# B&R Automation Studio project MappAssetInt
Automation Studio 4.12.9.18 SP; technology packages: mapp 5.24.2

## Configuration X20CP

CPU X20CP3687X, AutomationRuntime 6.7.6, Build 11.3.0, Safety 0.0, Vc 6.0.0

### Task classes (Cpu.sw)
```
Cyclic#8:
  AssetTest <- AssetTest.prg
  Sample <- exAssetInt.Sample.prg
  Shift <- Shift.prg
VcDataObjects: Vis <- Vis.dob
Binaries: vcnet, udbdef, vcrt, vcpkat, vcctext, vctcal, vcfile, vcgclass, vccstr, vcpdsw, arial, vcdsint, vcmgr, vcdsloc, vcfntttf, vccovl, vcshared, arialbd, vcalarm, vccdt, vcpdvnc, vcpfar00, vcbclass, TCData, vccnum, arsvcreg, vccshape, vccbtn, vccddbox, Vis01, Vis02, Vis03, vcclbox, vccpopup, arconfig, User, Config, ashwd, ashwac, Role, asfw, iomap, sysconf, vcpfx20, Visu01, Visu03, Visu02, Config_1
Libraries: AsBrStr, MpData, MpBase, MpAssetInt, MpCom, FileIO, DataObj, astime, brsystem, sys_lib, runtime, standard, vcresman, asieccon, ashw, AsIODiag, exAssetInt, IecCheck
```

### Hardware
```
X20CP3687X : X20CP3687X v1.8.0.0
  Connector IF2:
    ActivateDevice = 1
    Vnc1
    VncVcObjectName1 = Vis
    VncKeyMappingFile1 = VC\PS2-Keyboard.dis
    VncRefreshRate1 = 500
    ActivateSnmp = 2
  Connector IF3:
    DNAConfiguration = manual
    CycleTime = 2000
  ConfigurationID = MappAssetInt_X20CP1583
  UserPartitionSize = 16
  UserRamSize = 731936
  RemMemSize = 300000
  TimerDeviceType = EPLX2X
  TimerDevice = X20CP3687X.IF3
  TaskClassIdleTime = 2000
  Cyclic1Duration = 2000
  Cyclic8Stack = 20000
  FileDevice1
  FileDeviceName1 = ARsim
  FileDevicePath1 = C:\Temp\AssetInt
  FileDevice2
  FileDeviceName2 = USER_HD
  FileDevicePath2 = F:\
  FtpUser1
  FtpUsername1 = admin
  FtpUserPassword1 = WA9hSMBXiqkZliudaf2dLB8I5WaEURjKd6F9iexMfBQ=
  FtpUserSalt1 = wS51ak4d
  FTPAccessRight1 = 0
  ActivateOpcUa = 1
  OpcUaInformationModels_PV_Version = 1
```

## Logical view

Binary libraries used (declarations not repeated): operator, runtime, astime, AsIecCon, sys_lib, DataObj, brsystem, FileIO, AsBrStr, standard, AsIODiag, MpBase, MpAssetInt 5.24.6, MpCom, MpData 5.24.6

### Variables.var
```iecst
(*.-.-.-.-.---------------------------------------------------------------------------------------------------------------------------------------------------------------------------------*)
VAR
	Memory : ARRAY[0..19] OF exCoreInternalRecordType;
	TmpStr1 : STRING[80];
	TmpStr2 : STRING[80];
END_VAR
(*.-.-.-.-.---------------------------------------------------------------------------------------------------------------------------------------------------------------------------------*)
VAR
	AutoCount : BOOL; (*Start auto count*)
END_VAR
VAR CONSTANT
	AutoCountCycle : UINT := 1000; (*Auto count cycle in ms*)
END_VAR
VAR
	AutoCountTime : TON_10ms;
END_VAR
(*.-.-.-.-.---------------------------------------------------------------------------------------------------------------------------------------------------------------------------------*)
VAR
	AutoCreateJobs : BOOL; (*Auto create jobs*)
	AutoCreatePieceCnt : UDINT; (*Job piece counter*)
	AutoCreateJobsCnt : UDINT; (*Job name counter*)
	AutoCreateJobsNum : {REDUND_UNREPLICABLE} UDINT := 30; (*Pieces per job auto create*)
END_VAR
(*.-.-.-.-.---------------------------------------------------------------------------------------------------------------------------------------------------------------------------------*)
VAR
	GetDateTime : BOOL;
	SetDateTime : BOOL;
	RTCtime_struct : RTCtime_typ;
END_VAR
(*.-.-.-.-.---------------------------------------------------------------------------------------------------------------------------------------------------------------------------------*)
VAR
	TestBootCounter : UDINT;
	TestResult : ARRAY[1..9] OF TestResultEnum;
	TestCase : ARRAY[1..9] OF BOOL;
	TestState : ARRAY[1..9] OF USINT;
	TestIdle : ARRAY[1..9] OF UDINT;
	TesMyId : USINT;
END_VAR
(*.-.-.-.-.---------------------------------------------------------------------------------------------------------------------------------------------------------------------------------*)
VAR
	exAssetIntCoreAdr : {REDUND_UNREPLICABLE} UDINT;
	exAssetIntCoreLen : {REDUND_UNREPLICABLE} UDINT;
	exAssetIntCore_0 : REFERENCE TO exAssetIntCore;
END_VAR
```

### Library Logical/exAssetInt/exAssetInt (IEC, version 1.50.0)

#### MpAssetInt.typ
```iecst
(*File Version 1008*)
(*------------------------------------------------------------------------------------------------------------------------------------------------------------------------------------------------------------------------------------------------------------------------------------------------------------------------------------------------------*)
(*Internal type*)

TYPE
	exCoreInternalDataType : 	STRUCT
		RecordIndexUsed : ARRAY[0..CORE_EVENT_NUM_MAX]OF BOOL; (*Next record ID*)
		RecordIndex : UINT; (*Next record ID*)
		RecordData : exCoreInternalRecordType;
		State : exAssetIntStateEnum;
		StateError : exAssetIntStateEnum := exASSETINT_STATE_NONE;
		InitAfterBoot : BOOL;
		TimeLastCallShift : TIME;
		DiffLastCallShift : UDINT;
		TimeLastCallProduction : TIME;
		DiffLastCallProduction : UDINT;
		JobPieceCounterOld : UDINT;
		JobRejectCounterOld : UDINT;
		ShiftPieceCounterOld : UDINT;
		ShiftRejectCounterOld : UDINT;
		ShiftId : SINT;
		ShiftName : STRING[20];
		TmpStr1 : STRING[500];
		TmpStr2 : STRING[50];
		Downtime : exAssetIntDowntimeEnum;
		DowntimeReason : STRING[50];
		ProductionTotalTime : UDINT;
		CurrentTime : DTGetTime;
		PowerOffTime : DATE_AND_TIME;
		TimeOfDay : TIME_OF_DAY;
		ShiftTotalTimeStart : UDINT;
		StatsRefresh : TON_10ms;
		BackupTimer : TON_10ms;
		DirCreate_0 : DirCreate;
		CreateMemory : CreateMemory;
		ReadEventData : ReadEventData;
		WriteEventData : WriteEventData;
		ReadLinkData : ReadLinkData;
		WriteLinkData : WriteLinkData;
		ExportEventData : ExportEventData;
		x : UINT;
		y : UINT;
	END_STRUCT;
	exCoreInternalRecordType : 	STRUCT
		CRC : USINT;
		FileName : STRING[80]; (*ID of the event*)
		EventType : exCoreInternalRecordEnum;
		TimeStart : DATE_AND_TIME; (*Event start*)
		TimeEnd : DATE_AND_TIME; (*Event end*)
		ShiftName : STRING[20]; (*Shift name*)
		JobName : STRING[20]; (*Job name.*)
		TotalTime : exAssetIntTimeType; (*Total time since this job started*)
		ScheduledDowntime : exAssetIntTimeType; (*Scheduled downtime since this job started*)
		UnscheduledDowntime : exAssetIntTimeType; (*Unsheduled downtime since this job started*)
		Uptime : exAssetIntTimeType; (*Uptime since this job started*)
		NominalProductionTime : exAssetIntTimeType; (*Time of production at nominal speed since this job started*)
		GoodProductionTime : exAssetIntTimeType; (*Time of good production since this job started*)
		ScheduledDowntimeRate : REAL; (*Percentage of scheduled downtime [%] since this job started*)
		UnscheduledDowntimeRate : REAL; (*Percentage of unscheduled downtime [%] since this job started*)
		NominalProductionTimeRate : REAL; (*Percentage of nominal speed running time[%] since this job started*)
		TargetPieces : UDINT; (*Specifies the target quantity of products to be produced by the machine at nominal speed*)
		TotalPieces : UDINT; (*Counter for total products since this job started*)
		GoodPieces : UDINT; (*Counter for good products since this job started*)
		RejectPieces : UDINT; (*Counter for reject products since this job started*)
		BadPieceRate : REAL; (*Percentage of bad products [%] since this job started*)
		CurrentProductionRate : REAL; (*Production rate since this job started [products / h]*)
		CurrentUser : STRING[50]; (*Currently active user*)
		AdditionalData : STRING[EVENT_ADDITONAL_DATA_LEN]; (*Additional data information*)
	END_STRUCT;
	exCoreInternalRecordEnum :
		(
		RecordTypeJob := 0,
		RecordTypeShift := 1,
		RecordTypeNoShift := 2,
		RecordTypeUptime := 3,
		RecordTypeDowntimeScheduled := 4,
		RecordTypeDowntimeUnscheduled := 5,
		RecordTypeUserChange := 6,
		RecordTypeTimeline := 10
		);
	exCoreInternalExportEnum :
		(
		ExportTypeJob,
		ExportTypeShift,
		ExportTypeTimeline
		);
	exConfigInternalDataType : 	STRUCT
		State : exAssetIntStateEnum;
		StateError : exAssetIntStateEnum := exASSETINT_STATE_NONE;
		ReadConfiguration : ReadConfiguration;
		WriteConfiguration : WriteConfiguration;
	END_STRUCT;
	exUIInternalDataType : 	STRUCT
		RecordStart : DINT; (*Visible list is starting from this index*)
		RecordCount : UINT; (*Total number of items*)
		RecordCountOld : UINT; (*Old record number is required for DESC list*)
		RecordData : exCoreInternalRecordType;
		TimeSeconds : UDINT;
		TimeLongest : UDINT;
		SortingStartTimeOld : exAssetIntUISortingEnum := exASSETINT_SORTING_ASC;
		DT_TO_DTStructure_0 : DTStructure;
		x : UDINT;
		y : UDINT;
		State : exAssetIntStateEnum;
		StateError : exAssetIntStateEnum := exASSETINT_STATE_NONE;
	END_STRUCT;
	exAssetIntLinkType : 	STRUCT
		Version : USINT; (*Data structure version*)
		MemoryDb : UDINT; (*Database memory*)
		MemoryJob : UDINT; (*Job data memory*)
		MemoryShift : UDINT; (*Shift data memory*)
		MemoryTimeline : UDINT; (*Timeline data memory*)
		StatsLastCall : DTStructure; (*Date and time when the stats were last calculated*)
		Configuration : exAssetIntCoreConfigType; (*Configuration structure*)
		RecordCount : UINT; (*Number of total records*)
		IsCoreActive : BOOL; (*Core function block is ready*)
		RefreshJobUI : BOOL; (*Update job stats in UI*)
		RefreshShiftUI : BOOL; (*Update shift stats in UI*)
		RefreshTimelineUI : BOOL; (*Update timeline stats in UI*)
		ShiftStatistics : exAssetIntShiftStatisticsType; (*Current shift stats*)
		ShiftTotalTime : LREAL; (*Milliseconds the job is running*)
		ShiftDowntimeScheduled : UDINT; (*Milliseconds of scheduled downtime*)
		ShiftDowntimeUnscheduled : UDINT; (*Milliseconds of unscheduled downtime*)
		ShiftSecondsToEnd : UDINT;
		JobStatistics : exAssetIntJobStatisticsType; (*Current job stats*)
		JobTotalTime : LREAL; (*Milliseconds the job is running*)
		JobDowntimeScheduled : UDINT; (*Milliseconds of scheduled downtime*)
		JobDowntimeUnscheduled : UDINT; (*Milliseconds of unscheduled downtime*)
		ShiftId : SINT := -1; (*Index of shift configuration*)
		ProductionStateStart : DATE_AND_TIME; (*Current state beginning*)
		ProductionState : exAssetIntUIProductionStateEnum; (*Current state*)
		ProductionTotalTime : LREAL; (*Milliseconds the state is running*)
		ProductionUserName : STRING[50]; (*Currently active user*)
		ProductionShiftName : STRING[20]; (*ShiftName for this timeline*)
		ProductionJobName : STRING[20]; (*Job name for this timeline*)
		ProductionDowntime : exAssetIntDowntimeEnum; (*Downtime for this timeline*)
		ProductionDowntimeReason : STRING[50]; (*Donwtime reason for this timeline*)
	END_STRUCT;
END_TYPE

(*Enum type*)

TYPE
	exAssetIntStateEnum :
		(
		exASSETINT_STATE_INIT_1 := 1, (*Init state*)
		exASSETINT_STATE_INIT_2 := 2, (*Init state*)
		exASSETINT_STATE_INIT_3 := 3, (*Init state*)
		exASSETINT_STATE_INIT_4 := 4, (*Init state*)
		exASSETINT_STATE_INIT_5 := 5, (*Init state*)
		exASSETINT_STATE_IDLE := 10, (*Wait for command and collect data*)
		exASSETINT_STATE_STORE_EVENT := 20, (*Store new event data*)
		exASSETINT_STATE_EXPORT_EVENTS := 21, (*Export all events*)
		exASSETINT_STATE_UI_BUFFER := 30, (*Copy job data from global buffer to UI buffer*)
		exASSETINT_STATE_UI_DATA := 31, (*Generate UI data*)
		exASSETINT_STATE_SAVE_CFG := 40, (*Save configuration*)
		exASSETINT_STATE_LOAD_CFG := 41, (*Load configuration*)
		exASSETINT_STATE_SAVE_LINK := 50, (*Save internal data*)
		exASSETINT_STATE_LOAD_LINK := 51, (*Load internal data*)
		exASSETINT_STATE_ERROR := 90, (*Error state*)
		exASSETINT_STATE_NONE := 99 (*Empty state*)
		);
	exAssetIntLogLevelEnum :
		(
		exASSETINT_LOG_OFF := 0, (*Logging is disabled*)
		exASSETINT_LOG_ERROR := 1, (*Only log errors*)
		exASSETINT_LOG_INFO := 2, (*Also log information*)
		exASSETINT_LOG_ALL := 3 (*Log everything*)
		);
	exAssetIntBufferOffsets :
		(
		exASSETINT_BUFFER_MEMORY := 0
		);
	exAssetIntUIStatusEnum :
		(
		exASSETINT_UI_STATUS_IDLE := 0, (*Status: Idle, Waiting for command*)
		exASSETINT_UI_STATUS_UPDATE := 1, (*Status: Updating UIConnect structer*)
		exASSETINT_UI_STATUS_FILTER := 2 (*Status: Showing filter-dialog*)
		);
	exAssetIntMemoryEnum :
		(
		exASSETINT_MEM_DB := 0, (*Database memory*)
		exASSETINT_MEM_JOB := 1, (*Job working memory*)
		exASSETINT_MEM_SHIFT := 2, (*Shift working memory*)
		exASSETINT_MEM_TIMELINE := 3 (*Timeline working memory*)
		);
	exAssetIntDowntimeEnum :
		(
		exASSETINT_NO_DOWNTIME := 0, (*No downtime active = uptime*)
		exASSETINT_SCHEDULED_DOWNTIME := 1, (*Additional scheduled downtime (e.g. monthly maintenance)*)
		exASSETINT_UNSCHEDULED_DOWNTIME := 2 (*Unscheduled downtime (e.g. machine fault)*)
		);
	exComSeveritiesEnum :
		(
		exCOM_SEV_SUCCESS := 0, (*Success - no error*)
		exCOM_SEV_INFORMATIONAL := 1, (*Severity: Informational*)
		exCOM_SEV_WARNING := 2, (*Severity: Warning*)
		exCOM_SEV_ERROR := 3 (*Severity: Error*)
		);
END_TYPE

(*Config type*)

TYPE
	exAssetIntCoreConfigType : 	STRUCT
		CalculationTimeBase : UDINT := 1000; (*Cycle time for calculating the current production rate*)
		Shifts : ARRAY[0..4]OF exAssetIntShiftParType := [5(0)]; (*Shift schedule in detailed*)
		Export : exAssetIntExportType; (*Configuration for export*)
	END_STRUCT;
	exAssetIntExportType : 	STRUCT
		JobStatistics : BOOL := TRUE; (*Export the job statistics or not.*)
		JobStatisticsFileNamePattern : STRING[50] := 'JobStatistics_%Y_%m_%d_%H_%M.csv'; (*Pattern for export job statistics file.*)
		ShiftStatistics : BOOL := TRUE; (*Export the shift statistics or not.*)
		ShiftStatisticsFileNamePattern : STRING[50] := 'ShiftStatistics_%Y_%m_%d_%H_%M.csv'; (*Pattern for export shift statistics file.*)
		Timeline : BOOL := TRUE; (*Export the timeline statistics or not.*)
		TimelineFileNamePattern : STRING[50] := 'Timeline_%Y_%m_%d_%H_%M.csv'; (*Pattern for export timeline  file.*)
		TimestampPattern : STRING[50] := '%Y-%m-%d %H:%M:%S'; (*Timestamp pattern in exported file.*)
		DecimalDigits : UINT := 2; (*Specifies how many decimal positions are saved*)
		ColumnSeparator : STRING[1] := ','; (*Delimiter used to split up PVs in the .csv file*)
		DecimalMark : STRING[1] := '.'; (*Character to be used for the decimal separator*)
	END_STRUCT;
	exAssetIntShiftParType : 	STRUCT
		Name : STRING[20]; (*Shift name*)
		TotalTime : exAssetIntTimeSlotType; (*Total time of one shift*)
		ScheduledDowntime : ARRAY[0..9]OF exAssetIntScheduledDowntimeType; (*Scheduled downtime in one shift*)
	END_STRUCT;
	exAssetIntTimeSlotType : 	STRUCT
		Start : TIME_OF_DAY; (*Start time.*)
		End : TIME_OF_DAY; (*End time*)
	END_STRUCT;
	exAssetIntScheduledDowntimeType : 	STRUCT
		Reason : STRING[50]; (*Downtime reason*)
		Start : TIME_OF_DAY; (*Start time.*)
		End : TIME_OF_DAY; (*End time*)
	END_STRUCT;
END_TYPE

(*Parameter type*)

TYPE
	exAssetIntParType : 	STRUCT
		NominalProductionRate : REAL := 0.0; (*Nominal production rate [products / h]*)
		Job : STRING[20] := 'Job1'; (*Currently active production job*)
		CurrentUser : STRING[50]; (*Currently logged in user*)
		AdditionalData : STRING[255]; (*Additional data to be logged*)
	END_STRUCT;
END_TYPE

(*UI type*)

TYPE
	exAssetIntUITrendType : 	STRUCT
		SaexleData : ARRAY[0..365]OF REAL; (*FB->VC:Saexle data for trend data*)
		SaexleRate : UDINT; (*FB->VC:Saexle rate datapoint for trend data*)
		SaexleCount : UDINT; (*FB->VC:Saexle count datapoint for trend data*)
		SaexleDateTime : DATE_AND_TIME; (*FB->VC:Saexle DataTime datapoint for trend data*)
		MinValue : REAL; (*FB->VC:Min.value datapoint for trend data*)
		MaxValue : REAL; (*FB->VC:Max.value datapoint for trend data*)
		HideCurve : INT; (*FB->VC:Hide the curve if set to 1, status datapoint for trend curve*)
		TimeZoom : REAL; (*FB->VC:Zoom datapoint for trend time scale.*)
		TimeScroll : REAL; (*FB->VC:Scoll datapoint for trend time scale.*)
	END_STRUCT;
	exAssetIntUIShiftListType : 	STRUCT
		ShiftNames : ARRAY[0..5]OF STRING[20]; (*FB->VC: Shift names, *)
		SelectedIndex : UINT; (*VC->FB: Selection index for ShiftList.*)
		MaxSelection : USINT;
	END_STRUCT;
	exAssetIntTrendUIConnectType : 	STRUCT
		Status : exAssetIntUIStatusEnum; (*Status of UI function block*)
		ScheduledDowntimeRate : exAssetIntUITrendType; (*Trend for scheduled downtime rate*)
		UnscheduledDowntimeRate : exAssetIntUITrendType; (*Trend for unscheduled downtime rate*)
		NominalProductionRate : exAssetIntUITrendType; (*Trend for nominal production rate*)
		BadPieceRate : exAssetIntUITrendType; (*Trend for bad piece rate*)
		ShiftList : exAssetIntUIShiftListType; (*Determine which shift in the day is shown in the trend*)
		Filter : exAssetIntUIFilterType; (*Output filter.*)
	END_STRUCT;
	exAssetIntUITimelineOutputType : 	STRUCT
		StartTime : ARRAY[0..UI_TIMELINE_IDX]OF DATE_AND_TIME; (*FB->VC:Start time of this state*)
		ShiftName : ARRAY[0..UI_TIMELINE_IDX]OF STRING[20]; (*FB->VC:Shift name*)
		JobName : ARRAY[0..UI_TIMELINE_IDX]OF STRING[20]; (*FB->VC:Job name*)
		ProductionState : ARRAY[0..UI_TIMELINE_IDX]OF exAssetIntUIProductionStateEnum; (*FB->VC:Production state*)
		Reason : ARRAY[0..UI_TIMELINE_IDX]OF STRING[50]; (*FB->VC:Reason of this state*)
		Duration : ARRAY[0..UI_TIMELINE_IDX]OF exAssetIntTimeType; (*FB->VC:Duration of this state*)
		DurationBar : ARRAY[0..UI_TIMELINE_IDX]OF exAssetIntUITimeBargraphType; (*FB->VC:Duration of this state in a graphic way*)
		RangeStart : REAL; (*Displayed range: Start %*)
		RangeEnd : REAL; (*Displayed range: End %*)
		PageUp : BOOL; (*Command: Page Up (Scroll Up)*)
		StepUp : BOOL; (*Command: Line Up (Scroll Up)*)
		StepDown : BOOL; (*Command: Line Down (Scroll Down)*)
		PageDown : BOOL; (*Command: Page Down (Scroll Down)*)
	END_STRUCT;
	exAssetIntUITimeBargraphType : 	STRUCT
		Duration : UDINT; (*FB->VC:EndValue(lenth) of the scale*)
		Color : UDINT; (*FB->VC:ColorDatapoint of the scale*)
	END_STRUCT;
	exAssetIntTimelineUIConnectType : 	STRUCT
		Status : exAssetIntUIStatusEnum; (*Status of UI function block*)
		Output : exAssetIntUITimelineOutputType; (*Output information.*)
		Filter : exAssetIntUIFilterType; (*Output filter.*)
	END_STRUCT;
	exAssetIntTimeType : 	STRUCT
		Hours : UDINT; (*Numbers of hours*)
		Minutes : USINT; (*Numbers of minutes within an hour*)
		Seconds : USINT; (*Numbers of seconds within a minute*)
	END_STRUCT;
	exAssetIntShiftListUIConnectType : 	STRUCT
		Status : exAssetIntUIStatusEnum; (*Status of UI function block*)
		Output : exAssetIntUIShiftListOutputType; (*Output information.*)
		Filter : exAssetIntUIFilterType; (*Output filter.*)
	END_STRUCT;
	exAssetIntUIShiftListOutputType : 	STRUCT
		StartTime : ARRAY[0..UI_SHIFT_LIST_IDX]OF DATE_AND_TIME; (*Start time list*)
		EndTime : ARRAY[0..UI_SHIFT_LIST_IDX]OF DATE_AND_TIME; (*End time list*)
		ShiftName : ARRAY[0..UI_SHIFT_LIST_IDX]OF STRING[20]; (*Shift ID list*)
		CurrentUser : ARRAY[0..UI_SHIFT_LIST_IDX]OF STRING[50]; (*Currently active user*)
		AdditionalData : ARRAY[0..UI_SHIFT_LIST_IDX]OF STRING[255]; (*Additional data information*)
		TargetPieces : ARRAY[0..UI_SHIFT_LIST_IDX]OF UDINT; (*Target pieces list*)
		TotalPieces : ARRAY[0..UI_SHIFT_LIST_IDX]OF UDINT; (*Total pieces list*)
		GoodPieces : ARRAY[0..UI_SHIFT_LIST_IDX]OF UDINT; (*Good pieces list*)
		RejectPieces : ARRAY[0..UI_SHIFT_LIST_IDX]OF UDINT; (*Reject pieces list*)
		BadPieceRate : ARRAY[0..UI_SHIFT_LIST_IDX]OF REAL; (*bad piece rate list*)
		TotalTime : ARRAY[0..UI_SHIFT_LIST_IDX]OF exAssetIntTimeType; (*Total time list*)
		ScheduledDowntime : ARRAY[0..UI_SHIFT_LIST_IDX]OF exAssetIntTimeType; (*Scheduled Downtime list*)
		UnscheduledDowntime : ARRAY[0..UI_SHIFT_LIST_IDX]OF exAssetIntTimeType; (*Unscheduled Downtime list*)
		Uptime : ARRAY[0..UI_SHIFT_LIST_IDX]OF exAssetIntTimeType; (*Uptime list*)
		GoodProductionTime : ARRAY[0..UI_SHIFT_LIST_IDX]OF exAssetIntTimeType; (*Good production time list*)
		NominalProductionTime : ARRAY[0..UI_SHIFT_LIST_IDX]OF exAssetIntTimeType; (*nominal production time list*)
		NominalProductionRate : ARRAY[0..UI_SHIFT_LIST_IDX]OF REAL; (*nominal production rate list*)
		ShiftProductionRate : ARRAY[0..UI_SHIFT_LIST_IDX]OF REAL; (*Shift production rate list*)
		ScheduledDowntimeRate : ARRAY[0..UI_SHIFT_LIST_IDX]OF REAL; (*scheduled downtime rate list*)
		UnscheduledDowntimeRate : ARRAY[0..UI_SHIFT_LIST_IDX]OF REAL; (*unscheduled downtime rate list*)
		ProductionRate : ARRAY[0..UI_SHIFT_LIST_IDX]OF REAL; (*current production rate list*)
		RangeStart : REAL; (*Displayed range: Start %*)
		RangeEnd : REAL; (*Displayed range: End %*)
		PageUp : BOOL; (*Command: Page Up (Scroll Up)*)
		StepUp : BOOL; (*Command: Line Up (Scroll Up)*)
		StepDown : BOOL; (*Command: Line Down (Scroll Down)*)
		PageDown : BOOL; (*Command: Page Down (Scroll Down)*)
		IdealProductionRate : ARRAY[0..UI_SHIFT_LIST_IDX]OF REAL; (*ideal production rate list*)
		JobName : ARRAY[0..UI_SHIFT_LIST_IDX]OF STRING[20]; (*Job name list*)
	END_STRUCT;
	exAssetIntUIShiftListJobType : 	STRUCT  (*Jobs within one shift*)
		Name : ARRAY[0..9]OF STRING[20]; (*Name of the job*)
	END_STRUCT;
	exAssetIntListUISetupType : 	STRUCT
		ScrollWindow : USINT := 0; (*Scroll Window (overlap for PageUp/Down)*)
		SortingStartTime : exAssetIntUISortingEnum := exASSETINT_SORTING_DESC;
	END_STRUCT;
	exAssetIntJobListUIConnectType : 	STRUCT
		Status : exAssetIntUIStatusEnum; (*Status of UI function block*)
		Output : exAssetIntUIJobListOutputType; (*Output information.*)
		Filter : exAssetIntUIFilterType; (*Output filter.*)
	END_STRUCT;
	exAssetIntUIJobListOutputType : 	STRUCT
		JobStartTime : ARRAY[0..UI_JOB_LIST_IDX]OF DATE_AND_TIME; (*Job start time list*)
		JobEndTime : ARRAY[0..UI_JOB_LIST_IDX]OF DATE_AND_TIME; (*Job end time list*)
		JobName : ARRAY[0..UI_JOB_LIST_IDX]OF STRING[20]; (*Job name list*)
		CurrentUser : ARRAY[0..UI_JOB_LIST_IDX]OF STRING[50]; (*Currently active user*)
		AdditionalData : ARRAY[0..UI_JOB_LIST_IDX]OF STRING[255]; (*Additional data information*)
		TotalPieces : ARRAY[0..UI_JOB_LIST_IDX]OF UDINT; (*Total pieces list*)
		GoodPieces : ARRAY[0..UI_JOB_LIST_IDX]OF UDINT; (*Good pieces list*)
		RejectPieces : ARRAY[0..UI_JOB_LIST_IDX]OF UDINT; (*Reject pieces list*)
		BadPieceRate : ARRAY[0..UI_JOB_LIST_IDX]OF REAL; (*bad piece rate list*)
		TotalTime : ARRAY[0..UI_JOB_LIST_IDX]OF exAssetIntTimeType; (*Total time list*)
		ScheduledDowntime : ARRAY[0..UI_JOB_LIST_IDX]OF exAssetIntTimeType; (*Scheduled Downtime list*)
		UnscheduledDowntime : ARRAY[0..UI_JOB_LIST_IDX]OF exAssetIntTimeType; (*Unscheduled Downtime list*)
		Uptime : ARRAY[0..UI_JOB_LIST_IDX]OF exAssetIntTimeType; (*Uptime list*)
		GoodProductionTime : ARRAY[0..UI_JOB_LIST_IDX]OF exAssetIntTimeType; (*Good production time list*)
		NominalProductionTime : ARRAY[0..UI_JOB_LIST_IDX]OF exAssetIntTimeType; (*nominal production time list*)
		NominalProductionRate : ARRAY[0..UI_JOB_LIST_IDX]OF REAL; (*nominal production rate list*)
		ScheduledDowntimeRate : ARRAY[0..UI_JOB_LIST_IDX]OF REAL; (*scheduled downtime rate list*)
		UnscheduledDowntimeRate : ARRAY[0..UI_JOB_LIST_IDX]OF REAL; (*unscheduled downtime rate list*)
		ProductionRate : ARRAY[0..UI_JOB_LIST_IDX]OF REAL; (*current production rate list*)
		RangeStart : REAL; (*Displayed range: Start %*)
		RangeEnd : REAL; (*Displayed range: End %*)
		PageUp : BOOL; (*Command: Page Up (Scroll Up)*)
		StepUp : BOOL; (*Command: Line Up (Scroll Up)*)
		StepDown : BOOL; (*Command: Line Down (Scroll Down)*)
		PageDown : BOOL; (*Command: Page Down (Scroll Down)*)
		ShiftName : ARRAY[0..UI_JOB_LIST_IDX]OF STRING[20]; (*Shift ID list*)
	END_STRUCT;
	exAssetIntUISortingEnum :
		(
		exASSETINT_SORTING_ASC := 0, (*Sorting ascending*)
		exASSETINT_SORTING_DESC := 1 (*Sorting descending*)
		);
	exAssetIntUIProductionStateEnum :
		(
		exASSETINT_STATE_NO_SHIFT_ACTIVE := 0, (*Inactive state*)
		exASSETINT_STATE_UPTIME := 1, (*Uptime state*)
		exASSETINT_STATE_SCHDL_DOWNTIME := 2, (*Scheduled downtime state*)
		exASSETINT_STATE_UNSCH_DOWNTIME := 3, (*Unscheduled downtime state*)
		exASSETINT_STATE_USER_CHANGE := 4 (*User change*)
		);
	exAssetIntUICurrDTFilterType : 	STRUCT
		Enable : BOOL; (*Enable Filter*)
		DateTime : DATE_AND_TIME; (*Date and time of filter*)
	END_STRUCT;
	exAssetIntUISetDTFilterType : 	STRUCT
		Enable : BOOL; (*Enable Filter*)
		Year : UINT; (*Date&Time: Year*)
		Month : USINT; (*Date&Time: Month*)
		Day : USINT; (*Date&Time: Day*)
		Hour : USINT; (*Date&Time: Hour*)
		Minute : USINT; (*Date&Time: Minute*)
	END_STRUCT;
	exAssetIntUIFilterDialogType : 	STRUCT
		LayerStatus : UINT := UI_LAYER_HIDE; (*			Filter.Dialog.LayerStatus := UI_LAYER_HIDE;
*)
		From : exAssetIntUISetDTFilterType; (*Display entries from given date&time*)
		Until : exAssetIntUISetDTFilterType; (*Display entries until given date&time*)
		Confirm : BOOL;
		Cancel : BOOL;
	END_STRUCT;
	exAssetIntUIFilterType : 	STRUCT
		ShowDialog : BOOL;
		Dialog : exAssetIntUIFilterDialogType; (*Dialog-data to change filter-settings*)
		Current : exAssetIntUICurrentFilterType; (*Currently active filter settings*)
		DefaultLayerStatus : UINT;
	END_STRUCT;
	exAssetIntUICurrentFilterType : 	STRUCT
		From : exAssetIntUICurrDTFilterType; (*Starting time of current filter*)
		Until : exAssetIntUICurrDTFilterType; (*End time of current filter*)
	END_STRUCT;
END_TYPE

(*Info type*)

TYPE
	exAssetIntJobStatisticsType : 	STRUCT
		JobName : STRING[20]; (*Job name.*)
		StartTime : DATE_AND_TIME;
		TotalTime : exAssetIntTimeType; (*Total time since this job started*)
		ScheduledDowntime : exAssetIntTimeType; (*Scheduled downtime since this job started*)
		UnscheduledDowntime : exAssetIntTimeType; (*Unsheduled downtime since this job started*)
		Uptime : exAssetIntTimeType; (*Uptime since this job started*)
		NominalProductionTime : exAssetIntTimeType; (*Time of production at nominal speed since this job started*)
		GoodProductionTime : exAssetIntTimeType; (*Time of good production since this job started*)
		ScheduledDowntimeRate : REAL; (*Percentage of scheduled downtime [%] since this job started*)
		UnscheduledDowntimeRate : REAL; (*Percentage of unscheduled downtime [%] since this job started*)
		NominalProductionTimeRate : REAL; (*Percentage of nominal speed running time[%] since this job started*)
		TotalPieces : UDINT; (*Counter for total products since this job started*)
		GoodPieces : UDINT; (*Counter for good products since this job started*)
		RejectPieces : UDINT; (*Counter for reject products since this job started*)
		BadPieceRate : REAL; (*Percentage of bad products [%] since this job started*)
		CurrentProductionRate : REAL; (*Production rate since this job started [products / h]*)
		CurrentUser : STRING[50]; (*Currently active user*)
		AdditionalData : STRING[EVENT_ADDITONAL_DATA_LEN]; (*Additional data information*)
	END_STRUCT;
	exAssetIntShiftStatisticsType : 	STRUCT
		ShiftName : STRING[20]; (*Shift name.*)
		StartTime : DATE_AND_TIME;
		TotalTime : exAssetIntTimeType; (*Total time since this shift started*)
		ScheduledDowntime : exAssetIntTimeType; (*Scheduled downtime since this shift started*)
		UnscheduledDowntime : exAssetIntTimeType; (*Unsheduled downtime since this shift started*)
		Uptime : exAssetIntTimeType; (*Uptime since this shift started*)
		GoodProductionTime : exAssetIntTimeType; (*Time of good production since this shift started*)
		NominalProductionTime : exAssetIntTimeType; (*Time of production at nominal speed since this shift started*)
		ScheduledDowntimeRate : REAL; (*Percentage of scheduled downtime [%] since this shift started*)
		UnscheduledDowntimeRate : REAL; (*Percentage of unscheduled downtime [%] since this shift started*)
		NominalProductionTimeRate : REAL; (*Percentage of nominal speed running time[%] since this shift started*)
		TargetPieces : UDINT; (*Counter for target products since this shift started*)
		TotalPieces : UDINT; (*Counter for total products since this shift started*)
		GoodPieces : UDINT; (*Counter for good products since this shift started*)
		RejectPieces : UDINT; (*Counter for reject products since this shift started*)
		BadPieceRate : REAL; (*Percentage of bad products [%] since this shift started*)
		CurrentProductionRate : REAL; (*Production rate since this shift started [products / h]*)
		CurrentUser : STRING[50]; (*Currently active user*)
		AdditionalData : STRING[255]; (*Additional data information*)
		IdealProductionRate : REAL; (*Ideal production rate*)
	END_STRUCT;
	exAssetIntCoreInfoType : 	STRUCT
		ShiftStatistics : exAssetIntShiftStatisticsType; (*Shift statistics*)
		JobStatistics : exAssetIntJobStatisticsType; (*Job statistics*)
		Diag : exAssetIntDiagType; (*Additional diagnostic information*)
	END_STRUCT;
	exAssetIntInfoType : 	STRUCT
		Diag : exAssetIntDiagType; (*Additional diagnostic information*)
	END_STRUCT;
	exAssetIntDiagType : 	STRUCT
		StatusID : exAssetIntStatusIDType; (*Segmented StatusID output*)
	END_STRUCT;
	exAssetIntStatusIDType : 	STRUCT
		ID : exAssetIntErrorEnum; (*StatusID as enumerator*)
		Severity : exComSeveritiesEnum; (*Severity of the error*)
		Code : UINT; (*Error code*)
	END_STRUCT;
END_TYPE
```

#### Constants.var - Exported constants
```iecst
(*File Version 1007*)
(*------------------------------------------------------------------------------------------------------------------------------------------------------------------------------------------------------------------------------------------------------------------------------------------------------------------------------------------------------*)
(*General constants*)
(*------------------------------------------------------------------------------------------------------------------------------------------------------------------------------------------------------------------------------------------------------------------------------------------------------------------------------------------------------*)
VAR CONSTANT
	CORE_FOLDER_NAME : STRING[50] := 'AssetIntData'; (*Name of the event folder*)
	CORE_EVENT_NUM_MAX : UINT := 500; (*Maximum number of events*)
	CORE_BACKUP_TIMER : UINT := 10; (*Backup timer (minutes) for internal data*)
	EVENT_ADDITONAL_DATA_LEN : UINT := 100; (*Length of the event comment*)
	EXLINK_VERSION : USINT := 1; (*exLink structure version*)
END_VAR
(*------------------------------------------------------------------------------------------------------------------------------------------------------------------------------------------------------------------------------------------------------------------------------------------------------------------------------------------------------*)
(*Export constants*)
(*------------------------------------------------------------------------------------------------------------------------------------------------------------------------------------------------------------------------------------------------------------------------------------------------------------------------------------------------------*)
VAR CONSTANT
	EXPORT_BUFFER : UINT := 500; (*Length of the buffer for the event export*)
	EXPORT_JOB_TITEL : STRING[100] := 'AssetInt Job Statistics Export File'; (*Export file header*)
	EXPORT_SHIFT_TITEL : STRING[100] := 'AssetInt Shift Statistics Export File'; (*Export file header*)
	EXPORT_TIMELINE_TITEL : STRING[100] := 'AssetInt Timeline Statistics Export File'; (*Export file header*)
	EXPORT_JOB_HEADER : STRING[400] := 'Job Start Time;Job End Time;Job Name;Current User;Additional Data;Total Pieces;Good Pieces;Reject Pieces;Bad Piece Rate;Total Time;Scheduled Downtime;Unscheduled Downtime;Uptime;Good Production Time;Nominal Production Time;Nominal Production Time Rate;Scheduled Downtime Rate;Unscheduled Downtime Rate;Production Rate;Shift Name'; (*Export file column headers*)
	EXPORT_SHIFT_HEADER : STRING[400] := 'Job Start Time;Job End Time;Job Name;Current User;Additional Data;Total Pieces;Good Pieces;Reject Pieces;Bad Piece Rate;Total Time;Scheduled Downtime;Unscheduled Downtime;Uptime;Good Production Time;Nominal Production Time;Nominal Production Time Rate;Scheduled Downtime Rate;Unscheduled Downtime Rate;Production Rate;Shift Name'; (*Export file column headers*)
	EXPORT_TIMELINE_HEADER : STRING[400] := 'Start Time;Shift ID;Production State;Reason;Duration;Job Name'; (*Export file column headers*)
END_VAR
(*------------------------------------------------------------------------------------------------------------------------------------------------------------------------------------------------------------------------------------------------------------------------------------------------------------------------------------------------------*)
(*UI constants*)
(*------------------------------------------------------------------------------------------------------------------------------------------------------------------------------------------------------------------------------------------------------------------------------------------------------------------------------------------------------*)
VAR CONSTANT
	UI_SHIFT_LIST_IDX : UINT := 7; (*Max index for list box entries for shift data*)
	UI_TIMELINE_IDX : UINT := 7; (*Max index for list box entries for timeline data*)
	UI_JOB_LIST_IDX : UINT := 7; (*Max index for list box entries for job data*)
	UI_SHIFT_SHOW_JOBS : BOOL := FALSE; (*Show job changes in shift list*)
	UI_LAYER_SHOW : UINT := 0; (*Hide dialog layer*)
	UI_LAYER_HIDE : UINT := 1; (*Show dialog layer*)
	UI_LAYER_LOCK : UINT := 2; (*Lock dialog layer*)
END_VAR
(*------------------------------------------------------------------------------------------------------------------------------------------------------------------------------------------------------------------------------------------------------------------------------------------------------------------------------------------------------*)
(*Logger constants*)
(*------------------------------------------------------------------------------------------------------------------------------------------------------------------------------------------------------------------------------------------------------------------------------------------------------------------------------------------------------*)
VAR CONSTANT
	LOG_LEN : UINT := 100; (*Length of one log entry (minimum size is 50)*)
	LOG_NUM : UINT := 50; (*Number of log entries*)
	LOG_LEVEL : exAssetIntLogLevelEnum := exASSETINT_LOG_ALL; (*Define log level details*)
	CHAR_RETURN : USINT := 13; (*Carriage return*)
END_VAR
(*------------------------------------------------------------------------------------------------------------------------------------------------------------------------------------------------------------------------------------------------------------------------------------------------------------------------------------------------------*)
(*Error codes*)
(*------------------------------------------------------------------------------------------------------------------------------------------------------------------------------------------------------------------------------------------------------------------------------------------------------------------------------------------------------*)
VAR CONSTANT
	ERR_ASSET_LINK : DINT := -1064239102; (*Input exLink is 0 pointer*)
	ERR_ASSET_LINK_VERSION : DINT := 100001; (*exLink version is not compatible with backup data*)
	ERR_ASSET_LINK_SIZE : DINT := 100002; (*exLink backup data has wrong size*)
	ERR_ASSET_TEMP_MEMORY : DINT := -1064136704; (*No temporary memory available, make sure core function block is enabled*)
	ERR_ASSET_INF_WAIT_CORE_FB : DINT := 1083346949; (*This component can only become active if MpAssetIntCore is active.*)
	ERR_ASSET_READ_RECORD_SIZE : DINT := -2138009590; (*Record size is not correct during reading event data*)
	ERR_ASSET_READ_CRC : DINT := 100000; (*Record CRC error during reading event data*)
	ERR_ASSET_READ_FILE_NAME : DINT := 100003; (*File name in event folder does not match the expected event#<index> pattern*)
	ERR_ASSET_CONFIG : DINT := -1064239096; (*Configuration link is 0 pointer*)
	ERR_ASSET_CONFIG_SIZE : DINT := 100004; (*Configuration file has wrong size during reading*)
	ERR_ASSET_READ_BUFFER_FULL : DINT := 100005; (*More valid event files exist than fit into the record buffer, excess file was skipped*)
	ERR_ASSET_SHIFT_CALC : DINT := -1064239097; (*Invalid shift configured*)
END_VAR
```

#### exAssetInt.fun - Exported functions and function blocks
```iecst
(*File Version 1006*)
(*------------------------------------------------------------------------------------------------------------------------------------------------------------------------------------------------------------------------------------------------------------------------------------------------------------------------------------------------------*)

FUNCTION_BLOCK exAssetIntCore (*mapp function block which can be used for asset intensity calculation.*) (* $GROUP=mapp Services,$CAT=Asset Intensity,$GROUPICON=Icon_mapp.png,$CATICON=Icon_exOee.png *)
	VAR_INPUT
		exLink : REFERENCE TO exAssetIntLinkType; (*Incoming communication handle (mapp standard interface)*) (* *) (*#PAR#;*)
		Enable : BOOL; (*Enables/Disables the function block (mapp standard interface)*) (* *) (*#PAR#;*)
		ErrorReset : BOOL; (*Resets all function block errors (mapp standard interface)*) (* *) (*#PAR#;*)
		Parameters : REFERENCE TO exAssetIntParType; (*Function block parameters (mapp standard interface)*) (* *) (*#PAR#; *)
		Logger : UDINT;
		Configuration : REFERENCE TO exAssetIntCoreConfigType;
		Update : BOOL; (*Updates the parameters (mapp standard interface)*) (* *) (*#PAR#; *)
		Downtime : exAssetIntDowntimeEnum; (*The machine is in down time*) (* *) (*#CMD#; *)
		DowntimeReason : REFERENCE TO STRING[50]; (*The reason for down time*) (* *) (*#CMD#; *)
		PieceCounter : UDINT; (*Total pieces counter.*) (* *) (*#CMD#; *)
		RejectCounter : UDINT; (*Reject pieces counter*) (* *) (*#CMD#; *)
		DeviceName : REFERENCE TO STRING[50]; (*Address of the exported device name*) (* *) (*#CMD#; *)
		StorageName : REFERENCE TO STRING[50]; (*Address of the storage device name*) (* *) (*#CMD#; *)
		Export : BOOL; (*Export the saved information to file*) (* *) (*#CMD#; *)
		Reset : BOOL; (*Reset the data buffer*) (* *) (*#CMD#; *)
	END_VAR
	VAR_OUTPUT
		Active : BOOL; (*Function block is active (mapp standard interface)*) (* *) (*#PAR#;*)
		Error : BOOL; (*Indicates an error (mapp standard interface)*) (* *) (*#PAR#;*)
		StatusID : DINT; (*Error/Status information (mapp standard interface)*) (* *) (*#PAR#; *)
		UpdateDone : BOOL; (*Update of parameters done (mapp standard interface)*) (* *) (*#PAR#; *)
		CommandBusy : BOOL; (*Function block is busy processing a command*) (* *) (*#CMD#OPT#;*)
		CommandDone : BOOL; (*True if a command finshed successfully.*) (* *) (*#CMD#OPT#;*)
		CurrentProductionRate : REAL; (*Current production rate [products / h] based on calculation time base*) (* *) (*#CYC#*)
		ScheduledDowntimeRate : REAL; (*Percentage of scheduled downtime [%]*) (* *) (*#CYC#;*)
		UnscheduledDowntimeRate : REAL; (*Percentage of unscheduled downtime [%]*) (* *) (*#CYC#;*)
		NominalProductionTimeRate : REAL; (*Percentage of running time at nominal production speed [%]*) (* *) (*#CYC#;*)
		BadPieceRate : REAL; (*Percentage of bad products [%]*) (* *) (*#CYC#;*)
		ExportDone : BOOL; (*Export command was succesfuly finished*) (* *) (*#CMD#; *)
		Info : exAssetIntCoreInfoType; (*Provide any further useful information as function block output.(mapp standard interface)*) (* *) (*#CMD#; *)
	END_VAR
	VAR
		Internal : {REDUND_UNREPLICABLE} exCoreInternalDataType; (*Internal data*)
		zzEdge00000 : BOOL;
		zzEdge00001 : BOOL;
		zzEdge00002 : BOOL;
		zzEdge00003 : BOOL;
	END_VAR
END_FUNCTION_BLOCK

FUNCTION_BLOCK exAssetIntCoreConfig
	VAR_INPUT
		Enable : BOOL; (*Enables/Disables the function block (mapp standard interface)*) (* *) (*#PAR#;*)
		ErrorReset : BOOL; (*Resets all function block errors (mapp standard interface)*) (* *) (*#PAR#;*)
		DeviceName : REFERENCE TO STRING[30]; (*Address of the exported device name*) (* *) (*#CMD#; *)
		Configuration : REFERENCE TO exAssetIntCoreConfigType;
		Logger : UDINT;
		Load : {REDUND_UNREPLICABLE} BOOL; (* *) (* *) (*#PAR#;*)
		Save : BOOL; (* *) (* *) (*#PAR#;*)
	END_VAR
	VAR_OUTPUT
		Active : BOOL; (*Function block is active (mapp standard interface)*) (* *) (*#PAR#;*)
		Error : BOOL; (*Indicates an error (mapp standard interface)*) (* *) (*#PAR#;*)
		StatusID : DINT; (*Error/Status information (mapp standard interface)*) (* *) (*#PAR#; *)
		CommandBusy : BOOL; (*Function block is busy processing a command*) (* *) (*#CMD#OPT#;*)
		CommandDone : BOOL; (*True if a command finshed successfully.*) (* *) (*#CMD#OPT#;*)
		Info : exAssetIntInfoType; (*Provide any further useful information as function block output.(mapp standard interface)*) (* *) (*#CMD#; *)
	END_VAR
	VAR
		Internal : {REDUND_UNREPLICABLE} exConfigInternalDataType; (*Internal data*)
		zzEdge00000 : BOOL;
		zzEdge00001 : BOOL;
		zzEdge00002 : BOOL;
	END_VAR
END_FUNCTION_BLOCK

FUNCTION_BLOCK exAssetIntJobListUI (*mapp function block which can be used for showing job statistics in a list *)
	VAR_INPUT
		exLink : REFERENCE TO exAssetIntLinkType; (*Incoming communication handle (mapp standard interface)*) (* *) (*#PAR#;*)
		Enable : BOOL; (*Enables/Disables the function block (mapp standard interface)*) (* *) (*#PAR#;*)
		ErrorReset : BOOL; (*Resets all function block errors (mapp standard interface)*) (* *) (*#PAR#;*)
		Logger : UDINT;
		UISetup : exAssetIntListUISetupType; (*Setup UI connection - must be configured before enabling the FB*) (* *) (*#PAR#; *)
		UIConnect : REFERENCE TO exAssetIntJobListUIConnectType; (*Connection structure for VC4 User interface*) (* *) (*#CMD#; *)
	END_VAR
	VAR_OUTPUT
		Active : BOOL; (*Function block is active (mapp standard interface)*) (* *) (*#PAR#;*)
		Error : BOOL; (*Indicates an error (mapp standard interface)*) (* *) (*#PAR#;*)
		StatusID : DINT; (*Error/Status information (mapp standard interface)*) (* *) (*#PAR#; *)
		Info : exAssetIntInfoType; (*Provide any further useful information as function block output.(mapp standard interface)*) (* *) (*#CMD#; *)
	END_VAR
	VAR
		Internal : {REDUND_UNREPLICABLE} exUIInternalDataType; (*Internal data*)
		zzEdge00000 : BOOL;
	END_VAR
END_FUNCTION_BLOCK

FUNCTION_BLOCK exAssetIntShiftListUI (*mapp function block which can be used for showing shift statistics in a list *)
	VAR_INPUT
		exLink : REFERENCE TO exAssetIntLinkType; (*Incoming communication handle (mapp standard interface)*) (* *) (*#PAR#;*)
		Enable : BOOL; (*Enables/Disables the function block (mapp standard interface)*) (* *) (*#PAR#;*)
		ErrorReset : BOOL; (*Resets all function block errors (mapp standard interface)*) (* *) (*#PAR#;*)
		Logger : UDINT;
		UISetup : exAssetIntListUISetupType; (*Setup UI connection - must be configured before enabling the FB*) (* *) (*#PAR#; *)
		UIConnect : REFERENCE TO exAssetIntShiftListUIConnectType; (*Connection structure for VC4 User interface*) (* *) (*#CMD#; *)
	END_VAR
	VAR_OUTPUT
		Active : BOOL; (*Function block is active (mapp standard interface)*) (* *) (*#PAR#;*)
		Error : BOOL; (*Indicates an error (mapp standard interface)*) (* *) (*#PAR#;*)
		StatusID : DINT; (*Error/Status information (mapp standard interface)*) (* *) (*#PAR#; *)
		Info : exAssetIntInfoType; (*Provide any further useful information as function block output.(mapp standard interface)*) (* *) (*#CMD#; *)
	END_VAR
	VAR
		Internal : {REDUND_UNREPLICABLE} exUIInternalDataType; (*Internal data*)
		zzEdge00000 : BOOL;
	END_VAR
END_FUNCTION_BLOCK

FUNCTION_BLOCK exAssetIntTimelineUI (*mapp function block which can be used for showing timeline statistics in a list *)
	VAR_INPUT
		exLink : REFERENCE TO exAssetIntLinkType; (*Incoming communication handle (mapp standard interface)*) (* *) (*#PAR#;*)
		Enable : BOOL; (*Enables/Disables the function block (mapp standard interface)*) (* *) (*#PAR#;*)
		ErrorReset : BOOL; (*Resets all function block errors (mapp standard interface)*) (* *) (*#PAR#;*)
		Logger : UDINT;
		UISetup : exAssetIntListUISetupType; (*Setup UI connection - must be configured before enabling the FB*) (* *) (*#PAR#; *)
		UIConnect : REFERENCE TO exAssetIntTimelineUIConnectType; (*Connection structure for VC4 User interface*) (* *) (*#CMD#; *)
	END_VAR
	VAR_OUTPUT
		Active : BOOL; (*Function block is active (mapp standard interface)*) (* *) (*#PAR#;*)
		Error : BOOL; (*Indicates an error (mapp standard interface)*) (* *) (*#PAR#;*)
		StatusID : DINT; (*Error/Status information (mapp standard interface)*) (* *) (*#PAR#; *)
		Info : exAssetIntInfoType; (*Provide any further useful information as function block output.(mapp standard interface)*) (* *) (*#CMD#; *)
	END_VAR
	VAR
		Internal : {REDUND_UNREPLICABLE} exUIInternalDataType; (*Internal data*)
		zzEdge00000 : BOOL;
	END_VAR
END_FUNCTION_BLOCK

FUNCTION_BLOCK CreateMemory
	VAR_INPUT
		Enable : BOOL;
		Size : UDINT;
		Logger : {REDUND_UNREPLICABLE} UDINT; (*Address of log buffer*)
	END_VAR
	VAR_OUTPUT
		MemoryDb : UDINT;
		MemoryJob : UDINT;
		MemoryShift : UDINT;
		MemoryTimeline : UDINT;
		Status : DINT;
	END_VAR
	VAR
		DatObjCreate_0 : DatObjCreate;
		MemoryType : exAssetIntMemoryEnum;
		TmpStr1 : STRING[100];
		TmpStr2 : STRING[100];
		Cnt : USINT;
		State : USINT;
	END_VAR
END_FUNCTION_BLOCK

FUNCTION_BLOCK ReadConfiguration
	VAR_INPUT
		Enable : BOOL;
		Device : REFERENCE TO STRING[50];
		Logger : {REDUND_UNREPLICABLE} UDINT; (*Address of log buffer*)
		Configuration : exAssetIntCoreConfigType;
	END_VAR
	VAR_OUTPUT
		Status : DINT;
	END_VAR
	VAR
		FileOpen_0 : FileOpen;
		FileClose_0 : FileClose;
		FileRead_0 : FileRead;
		State : USINT;
	END_VAR
END_FUNCTION_BLOCK

FUNCTION_BLOCK WriteConfiguration
	VAR_INPUT
		Enable : BOOL;
		Device : REFERENCE TO STRING[50];
		Logger : UDINT; (*Address of log buffer*)
		Configuration : exAssetIntCoreConfigType;
	END_VAR
	VAR_OUTPUT
		Status : DINT;
	END_VAR
	VAR
		FileCreate_0 : FileCreate;
		FileOpen_0 : FileOpen;
		FileClose_0 : FileClose;
		FileWrite_0 : FileWrite;
		Ident : UDINT;
		State : USINT;
	END_VAR
END_FUNCTION_BLOCK

FUNCTION_BLOCK ReadLinkData
	VAR_INPUT
		Enable : BOOL;
		Device : REFERENCE TO STRING[50];
		Logger : {REDUND_UNREPLICABLE} UDINT;
		Link : REFERENCE TO exAssetIntLinkType;
	END_VAR
	VAR_OUTPUT
		Status : DINT;
	END_VAR
	VAR
		FileOpen_0 : FileOpen;
		FileClose_0 : FileClose;
		FileRead_0 : FileRead;
		FileDelete_0 : FileDelete;
		LinkRead : exAssetIntLinkType;
		StatusRead : DINT;
		State : USINT;
	END_VAR
END_FUNCTION_BLOCK

FUNCTION_BLOCK WriteLinkData
	VAR_INPUT
		Enable : BOOL;
		Device : REFERENCE TO STRING[50];
		Logger : UDINT;
		Link : REFERENCE TO exAssetIntLinkType;
	END_VAR
	VAR_OUTPUT
		Status : DINT;
	END_VAR
	VAR
		FileCreate_0 : FileCreate;
		FileOpen_0 : FileOpen;
		FileClose_0 : FileClose;
		FileWrite_0 : FileWrite;
		Ident : UDINT;
		State : USINT;
	END_VAR
END_FUNCTION_BLOCK

FUNCTION_BLOCK ReadEventData
	VAR_INPUT
		Enable : BOOL;
		Device : STRING[50];
		Logger : {REDUND_UNREPLICABLE} UDINT;
		Memory : UDINT;
		RecordIndexUsed : REFERENCE TO ARRAY[0..CORE_EVENT_NUM_MAX] OF BOOL;
	END_VAR
	VAR_OUTPUT
		RecordCount : UINT;
		Status : DINT;
	END_VAR
	VAR
		DirOpen_0 : DirOpen;
		DirReadEx_0 : DirReadEx;
		DirClose_0 : DirClose;
		FileOpen_0 : FileOpen;
		FileClose_0 : FileClose;
		FileRead_0 : FileRead;
		FileDelete_0 : FileDelete;
		FileName : STRING[100];
		FileInfo_0 : fiDIR_READ_EX_DATA;
		RecordData : exCoreInternalRecordType;
		FirstEntryTime : DATE_AND_TIME;
		LastEntryTime : DATE_AND_TIME;
		FirstEntryRecord : UINT;
		LastEntryRecord : UINT;
		TmpStr1 : STRING[100];
		FileIndex : UINT;
		FileIndexCheck : DINT;
		NextFileNameGet : BOOL;
		NextFileNameReady : BOOL;
		Override : {REDUND_UNREPLICABLE} USINT;
		State : USINT;
		CRC : USINT;
		StatusRead : DINT;
		zzEdge00000 : BOOL;
	END_VAR
END_FUNCTION_BLOCK

FUNCTION_BLOCK WriteEventData
	VAR_INPUT
		Enable : BOOL;
		Device : STRING[50];
		Logger : UDINT; (*Address of log buffer*)
		RecordData : UDINT;
		RecordIndex : UINT;
	END_VAR
	VAR_OUTPUT
		Status : DINT;
	END_VAR
	VAR
		FileCreate_0 : FileCreate;
		FileOpen_0 : FileOpen;
		FileClose_0 : FileClose;
		FileWrite_0 : FileWrite;
		RecordDataIntern : exCoreInternalRecordType;
		TmpStr1 : STRING[100];
		TmpStr2 : STRING[10];
		Ident : UDINT;
		State : USINT;
		zzEdge00000 : BOOL;
	END_VAR
END_FUNCTION_BLOCK

FUNCTION_BLOCK ExportEventData
	VAR_INPUT
		Enable : BOOL;
		Device : STRING[50];
		Logger : UDINT; (*Address of log buffer*)
		RecordCount : UDINT;
		Memory : UDINT;
		Configuration : exAssetIntExportType;
	END_VAR
	VAR_OUTPUT
		Status : DINT;
	END_VAR
	VAR
		ExportType : exCoreInternalExportEnum;
		FileDelete_0 : FileDelete;
		FileCreate_0 : FileCreate;
		FileClose_0 : FileClose;
		FileWrite_0 : FileWrite;
		RtcGettime : {REDUND_UNREPLICABLE} RTCtime_typ;
		RecordDataIntern : exCoreInternalRecordType;
		DTStructure_0 : DTStructure;
		FileName : STRING[54]; (*+4 bytes to absorb %Y expansion from 2 to 4 chars*)
		TmpStr1 : STRING[54]; (*+4 bytes to absorb %Y expansion from 2 to 4 chars*)
		TmpStr2 : STRING[50];
		lrealStr : {REDUND_UNREPLICABLE} LREAL;
		Buffer : STRING[EXPORT_BUFFER];
		Offset : UDINT;
		idx : UDINT;
		State : USINT;
	END_VAR
END_FUNCTION_BLOCK

FUNCTION exAssetIntFilterListUI : UDINT
	VAR_INPUT
		Filter : REFERENCE TO exAssetIntUIFilterType;
		Status : REFERENCE TO exAssetIntUIStatusEnum;
		Logger : UDINT;
		State : exAssetIntStateEnum;
	END_VAR
	VAR
		DT_TO_DTStructure_0 : DTStructure;
	END_VAR
END_FUNCTION

FUNCTION exAssetIntScrollListUI : exAssetIntStateEnum
	VAR_INPUT
		RecordCount : UINT;
		ListMaxCount : UINT;
		PageUp : REFERENCE TO BOOL; (* *) (* *) (*#PAR#;*)
		PageDown : REFERENCE TO BOOL; (* *) (* *) (*#PAR#;*)
		StepUp : REFERENCE TO BOOL; (* *) (* *) (*#PAR#;*)
		StepDown : REFERENCE TO BOOL; (* *) (* *) (*#PAR#;*)
		RecordStart : REFERENCE TO DINT;
		RangeStart : REFERENCE TO REAL;
		RangeEnd : REFERENCE TO REAL;
		State : exAssetIntStateEnum;
	END_VAR
END_FUNCTION

FUNCTION exAssetIntBufferUI : UINT
	VAR_INPUT
		Memory : UDINT;
		exLink : exAssetIntLinkType; (*Incoming communication handle (mapp standard interface)*) (* *) (*#PAR#;*)
		SortingStartTime : exAssetIntUISortingEnum;
		Filter : exAssetIntUIFilterType;
		EventType : exCoreInternalRecordEnum;
	END_VAR
	VAR
		RecordData : exCoreInternalRecordType;
		RecordCount : UINT;
		y : UDINT;
	END_VAR
END_FUNCTION

FUNCTION exAssetIntFilterReset : BOOL
	VAR_INPUT
		Filter : REFERENCE TO exAssetIntUIFilterType;
	END_VAR
END_FUNCTION

FUNCTION exAssetIntCheckPreq : BOOL
	VAR_INPUT
		exLink : exAssetIntLinkType; (*Incoming communication handle (mapp standard interface)*) (* *) (*#PAR#;*)
		UIConnect : UDINT; (* *) (* *) (*#PAR#;*)
		Logger : UDINT;
		State : REFERENCE TO exAssetIntStateEnum;
		StatusID : REFERENCE TO DINT;
		InfoDiagStatusID : REFERENCE TO exAssetIntStatusIDType;
	END_VAR
END_FUNCTION

FUNCTION exAssetIntCheckShiftData : BOOL
	VAR_INPUT
		Configuration : exAssetIntCoreConfigType;
		Logger : UDINT;
		State : REFERENCE TO exAssetIntStateEnum;
		StatusID : REFERENCE TO DINT;
		InfoDiagStatusID : REFERENCE TO exAssetIntStatusIDType;
	END_VAR
	VAR
		TmpStr1 : STRING[100];
		TmpStr2 : STRING[100];
		y : USINT;
		x : USINT;
	END_VAR
END_FUNCTION

FUNCTION InsertEventData : USINT
	VAR_INPUT
		Memory : UDINT;
		RecordCount : UINT;
		RecordData : exCoreInternalRecordType;
	END_VAR
	VAR
		RecordMemory : REFERENCE TO exCoreInternalRecordType;
		sort : UDINT;
		x : INT;
		y : INT;
	END_VAR
END_FUNCTION

FUNCTION CreateLoggerEntry : USINT
	VAR_INPUT
		LogLevel : exAssetIntLogLevelEnum; (*Log Level*)
		LogMsg : UDINT; (*Log message*)
		LogBuffer : UDINT; (*Address of log buffer*)
	END_VAR
	VAR
		RtcGettime : RTCtime_typ;
		TmpStr : STRING[20];
		LastMsg : STRING[LOG_LEN];
		TmpMsg : STRING[LOG_LEN];
	END_VAR
END_FUNCTION

FUNCTION CreateErrorState : DINT
	VAR_INPUT
		ErrorID : DINT;
		ErrorMsg : UDINT;
		Logger : UDINT;
		Severity : exComSeveritiesEnum;
		State : REFERENCE TO exAssetIntStateEnum;
		DiagStatusID : REFERENCE TO exAssetIntStatusIDType;
	END_VAR
END_FUNCTION

FUNCTION CalcStatsJob : USINT
	VAR_INPUT
		exLink : exAssetIntLinkType; (*Incoming communication handle (mapp standard interface)*) (* *) (*#PAR#;*)
		DiffLastCall : UDINT;
		Downtime : exAssetIntDowntimeEnum;
		Parameter : exAssetIntParType;
		JobStatistics : REFERENCE TO exAssetIntJobStatisticsType;
	END_VAR
	VAR
		JobTotalTime : UDINT;
		Uptime : UDINT;
		NominalProductionTime : UDINT;
		GoodProductionTime : UDINT;
	END_VAR
END_FUNCTION

FUNCTION TrackShiftChange : BOOL
	VAR_INPUT
		exLink : REFERENCE TO exAssetIntLinkType; (*Incoming communication handle (mapp standard interface)*) (* *) (*#PAR#;*)
		Internal : REFERENCE TO exCoreInternalDataType; (*Internal data*)
		Info : REFERENCE TO exAssetIntCoreInfoType; (* *) (* *) (*#PAR#; *)
		Parameters : exAssetIntParType; (* *) (* *) (*#PAR#; *)
		Logger : UDINT;
	END_VAR
	VAR
		DiffTime : DINT;
	END_VAR
END_FUNCTION

FUNCTION TrackProductionState : BOOL
	VAR_INPUT
		exLink : REFERENCE TO exAssetIntLinkType; (*Incoming communication handle (mapp standard interface)*) (* *) (*#PAR#;*)
		Internal : REFERENCE TO exCoreInternalDataType; (*Internal data*)
		Parameters : exAssetIntParType; (* *) (* *) (*#PAR#; *)
		Logger : UDINT;
	END_VAR
END_FUNCTION

FUNCTION CalcStatsShift : USINT
	VAR_INPUT
		exLink : exAssetIntLinkType; (*Incoming communication handle (mapp standard interface)*) (* *) (*#PAR#;*)
		DiffLastCall : UDINT;
		Downtime : exAssetIntDowntimeEnum;
		Parameter : exAssetIntParType;
		ShiftStatistics : REFERENCE TO exAssetIntShiftStatisticsType;
	END_VAR
	VAR
		ShiftTotalTime : UDINT;
		Uptime : UDINT;
		NominalProductionTime : UDINT;
		GoodProductionTime : UDINT;
	END_VAR
END_FUNCTION

FUNCTION CalcCrc : USINT
	VAR_INPUT
		data : UDINT;
		length : UINT;
	END_VAR
	VAR
		idx : UINT;
		_byte : USINT;
	END_VAR
END_FUNCTION

FUNCTION FindInstr : UDINT
	VAR_INPUT
		string1 : UDINT;
		string2 : UDINT;
	END_VAR
	VAR
		idx : UDINT;
	END_VAR
END_FUNCTION

FUNCTION ReplaceString : USINT
	VAR_INPUT
		dataSTR : UDINT;
		searchSTR : UDINT;
		replaceSTR : UDINT;
	END_VAR
	VAR
		idx : UDINT;
	END_VAR
END_FUNCTION

FUNCTION ReplaceDateTime : USINT
	VAR_INPUT
		dataSTR : UDINT;
		searchSTR : UDINT;
		value : UINT;
	END_VAR
	VAR
		lrealStr : LREAL;
	END_VAR
END_FUNCTION

FUNCTION NormalizeDateTime : LREAL
	VAR_INPUT
		value : UDINT;
	END_VAR
	VAR
		TmpStr1 : STRING[6] := '';
		TmpStr2 : STRING[6] := '';
	END_VAR
END_FUNCTION

FUNCTION NormalizeFloat : LREAL
	VAR_INPUT
		value : REAL;
		output : UDINT;
		configuration : exAssetIntExportType;
	END_VAR
	VAR
		idx : UDINT;
		tmpStr : STRING[50];
	END_VAR
END_FUNCTION
```

#### exAssetIntCore.st
```iecst
// -------------------------------------------------------------------------------------------
// File version 1013
// -------------------------------------------------------------------------------------------
// Core function block
FUNCTION_BLOCK exAssetIntCore
	// -------------------------------------------------------------------------------------------
	// Reset everything when enable is false
	IF NOT Enable THEN
		Active := FALSE;
		exLink.IsCoreActive := FALSE;
		StatusID := ERR_FUB_ENABLE_FALSE;
		Internal.State := exASSETINT_STATE_INIT_1;
		CreateLoggerEntry(exASSETINT_LOG_INFO, ADR('function block disabled'), Logger);
		RETURN;
	END_IF

	// Permanent watch critical values
	IF Internal.State <> exASSETINT_STATE_ERROR THEN
		// Make sure we have remanent buffer
		IF ADR(exLink) = 0 THEN
			// Set status, remember state, go to error state
			StatusID := CreateErrorState(ERR_ASSET_LINK, ADR('ERR: exLink is 0'), Logger, exCOM_SEV_ERROR, ADR(Internal.State), ADR(Info.Diag.StatusID));
			RETURN;
		END_IF
		// Make sure we have valid memory data
		IF (exLink.MemoryDb = 0 OR exLink.MemoryJob = 0 OR exLink.MemoryShift = 0 OR exLink.MemoryTimeline = 0) AND Active THEN
			// Set status, remember state, go to error state
			StatusID := CreateErrorState(ERR_ASSET_LINK, ADR('ERR: memory address is 0'), Logger, exCOM_SEV_ERROR, ADR(Internal.State), ADR(Info.Diag.StatusID));
			RETURN;
		END_IF
		// Make sure we have a configuration
		IF ADR(Configuration) = 0 THEN
			// Set status, remember state, go to error state
			StatusID := CreateErrorState(ERR_ASSET_LINK, ADR('ERR: No configuation attached'), Logger, exCOM_SEV_ERROR, ADR(Internal.State), ADR(Info.Diag.StatusID));
			RETURN;
		END_IF
		// Make sure we have a parameters
		IF ADR(Parameters) = 0 THEN
			// Set status, remember state, go to error state
			StatusID := CreateErrorState(ERR_ASSET_LINK, ADR('ERR: No parameters attached'), Logger, exCOM_SEV_ERROR, ADR(Internal.State), ADR(Info.Diag.StatusID));
			RETURN;
		END_IF
		// Make sure we have a device name
		IF ADR(DeviceName) = 0 THEN
			// Set status, remember state, go to error state
			StatusID := CreateErrorState(ERR_ASSET_LINK, ADR('ERR: No device name attached'), Logger, exCOM_SEV_ERROR, ADR(Internal.State), ADR(Info.Diag.StatusID));
			RETURN;
		END_IF
		// Make sure we have a storage name
		IF ADR(StorageName) = 0 THEN
			// Set status, remember state, go to error state
			StatusID := CreateErrorState(ERR_ASSET_LINK, ADR('ERR: No storage name attached'), Logger, exCOM_SEV_ERROR, ADR(Internal.State), ADR(Info.Diag.StatusID));
			RETURN;
		END_IF
	END_IF

	CASE Internal.State OF

		// -------------------------------------------------------------------------------------------
		// Wait for enable
		// -------------------------------------------------------------------------------------------
		exASSETINT_STATE_INIT_1:
			IF Enable THEN
				CreateLoggerEntry(exASSETINT_LOG_INFO, ADR('function block enabled'), Logger);

				exLink.RecordCount := 0;
				exLink.Version := EXLINK_VERSION;

				// -------------------------------------------------------------------------------------------
				// Reset error, status and function and internal blocks
				brsmemset(ADR(Info.Diag), 0, SIZEOF(Info.Diag));
				Error := FALSE;
				StatusID := ERR_OK;
				Internal.CreateMemory(Enable := FALSE);
				Internal.ReadEventData(Enable := FALSE);
				Internal.WriteEventData(Enable := FALSE);
				Internal.ReadEventData(Enable := FALSE);
				Internal.WriteEventData(Enable := FALSE);
				Internal.DirCreate_0.enable := FALSE;
				Internal.DirCreate_0();

				// Update time information
				Internal.CurrentTime(enable := TRUE);
				IF exLink.StatsLastCall.year > 0 THEN
					// Make sure we power back on in the future
					IF DiffDT(Internal.CurrentTime.DT1, DTStructure_TO_DT(ADR(exLink.StatsLastCall))) <> 16#FFFFFFFF THEN
						Internal.PowerOffTime := DTStructure_TO_DT(ADR(exLink.StatsLastCall));
					END_IF
				END_IF

				// -------------------------------------------------------------------------------------------
				// Create folder structure and read event data only after boot
				IF Internal.InitAfterBoot THEN
					Internal.State := exASSETINT_STATE_INIT_4;
				ELSE
					// -------------------------------------------------------------------------------------------
					// Try to restore backup when link data is empty
					IF exLink.MemoryDb = 0 THEN
						Internal.State := exASSETINT_STATE_LOAD_LINK;
					ELSE
						Internal.State := exASSETINT_STATE_INIT_2;
					END_IF
				END_IF
			END_IF

			// -------------------------------------------------------------------------------------------
			// Create folder structure
			// -------------------------------------------------------------------------------------------
		exASSETINT_STATE_INIT_2:
			Internal.DirCreate_0.enable := TRUE;
			Internal.DirCreate_0.pDevice := ADR(StorageName);
			Internal.DirCreate_0.pName := ADR(CORE_FOLDER_NAME);
			Internal.DirCreate_0();

			// -------------------------------------------------------------------------------------------
			// Folder structure successful created
			IF Internal.DirCreate_0.status = ERR_OK OR Internal.DirCreate_0.status = fiERR_DIR_ALREADY_EXIST THEN
				CreateLoggerEntry(exASSETINT_LOG_INFO, ADR('create folder structure ok'), Logger);
				Internal.State := exASSETINT_STATE_INIT_3;

				// Error
			ELSIF Internal.DirCreate_0.status <> ERR_FUB_BUSY THEN
				// Set status, remember state, go to error state
				StatusID := CreateErrorState(Internal.DirCreate_0.status, ADR('ERR: create folder structure'), Logger, exCOM_SEV_ERROR, ADR(Internal.State), ADR(Info.Diag.StatusID));
			END_IF

			// -------------------------------------------------------------------------------------------
			// Create internal memory
			// -------------------------------------------------------------------------------------------
		exASSETINT_STATE_INIT_3:
			Internal.CreateMemory.Enable := TRUE;
			Internal.CreateMemory.Size := CORE_EVENT_NUM_MAX*SIZEOF(Internal.RecordData);
			Internal.CreateMemory.Logger := Logger;
			Internal.CreateMemory();

			// -------------------------------------------------------------------------------------------
			// Memory structure successful created
			IF Internal.CreateMemory.Status = ERR_OK THEN
				CreateLoggerEntry(exASSETINT_LOG_INFO, ADR('create internal memory ok'), Logger);
				exLink.MemoryDb := Internal.CreateMemory.MemoryDb;
				exLink.MemoryJob := Internal.CreateMemory.MemoryJob;
				exLink.MemoryShift := Internal.CreateMemory.MemoryShift;
				exLink.MemoryTimeline := Internal.CreateMemory.MemoryTimeline;
				Internal.InitAfterBoot := TRUE;
				Internal.State := exASSETINT_STATE_INIT_4;

				// Error
			ELSIF Internal.CreateMemory.Status <> ERR_FUB_BUSY THEN
				// Set status, remember state, go to error state
				StatusID := CreateErrorState(Internal.CreateMemory.Status, ADR('ERR: create internal memory'), Logger, exCOM_SEV_ERROR, ADR(Internal.State), ADR(Info.Diag.StatusID));
			END_IF

			// -------------------------------------------------------------------------------------------
			// Read event data
			// -------------------------------------------------------------------------------------------
		exASSETINT_STATE_INIT_4:
			Internal.ReadEventData.Enable := TRUE;
			Internal.ReadEventData.Device := StorageName;
			Internal.ReadEventData.Memory := exLink.MemoryDb;
			Internal.ReadEventData.RecordIndexUsed := ADR(Internal.RecordIndexUsed);
			Internal.ReadEventData.Logger := Logger;
			Internal.ReadEventData();

			// Read events successful
			IF Internal.ReadEventData.Status = ERR_OK THEN
				CreateLoggerEntry(exASSETINT_LOG_INFO, ADR('read stored events ok'), Logger);

				// -------------------------------------------------------------------------------------------
				// Get record count, calculate next entry
				exLink.RecordCount := Internal.ReadEventData.RecordCount;
				Internal.State := exASSETINT_STATE_INIT_5;

				// Error
			ELSIF Internal.ReadEventData.Status <> ERR_FUB_BUSY THEN
				// Set status, remember state, go to error state
				StatusID := CreateErrorState(Internal.ReadEventData.Status, ADR('ERR: read stored events'), Logger, exCOM_SEV_ERROR, ADR(Internal.State), ADR(Info.Diag.StatusID));
			END_IF

			// -------------------------------------------------------------------------------------------
			// Set inital values
			// -------------------------------------------------------------------------------------------
		exASSETINT_STATE_INIT_5:
			// -------------------------------------------------------------------------------------------
			// Transfer start values
			exLink.JobStatistics.JobName := Parameters.Job;
			exLink.JobStatistics.CurrentUser := Parameters.CurrentUser;
			exLink.JobStatistics.AdditionalData := Parameters.AdditionalData;
			Internal.JobPieceCounterOld := PieceCounter;
			Internal.JobRejectCounterOld := RejectCounter;

			exLink.ShiftStatistics.CurrentUser := Parameters.CurrentUser;
			exLink.ShiftStatistics.AdditionalData := Parameters.AdditionalData;
			Internal.ShiftPieceCounterOld := PieceCounter;
			Internal.ShiftRejectCounterOld := RejectCounter;

			// -------------------------------------------------------------------------------------------
			// Check shift configuration for errors
			IF NOT exAssetIntCheckShiftData(Configuration, Logger, ADR(Internal.State), ADR(StatusID), ADR(Info.Diag.StatusID)) THEN
				RETURN;
			END_IF

			// Transfer configuration
			brsmemcpy(ADR(exLink.Configuration), ADR(Configuration), SIZEOF(Configuration));

			// -------------------------------------------------------------------------------------------
			// Remember start called time
			Internal.TimeLastCallShift := clock_ms();
			Internal.TimeLastCallProduction := clock_ms();

			// -------------------------------------------------------------------------------------------
			// Refresh UI data, finish up
			exLink.RefreshJobUI := TRUE;
			exLink.RefreshShiftUI := TRUE;
			exLink.RefreshTimelineUI := TRUE;
			Internal.State := exASSETINT_STATE_IDLE;

			// -------------------------------------------------------------------------------------------
			// Wait for new event
			// -------------------------------------------------------------------------------------------
		exASSETINT_STATE_IDLE:
			// Set core active, reset read write function blocks
			Active := TRUE;
			exLink.IsCoreActive := TRUE;
			Internal.ReadEventData(Enable := FALSE);
			Internal.WriteEventData(Enable := FALSE);

			// Update time information
			Internal.CurrentTime(enable := TRUE);
			DT_TO_DTStructure(Internal.CurrentTime.DT1, ADR(exLink.StatsLastCall));
			Internal.TimeOfDay := UDINT_TO_TOD((USINT_TO_UDINT(exLink.StatsLastCall.hour) * 3600000) + (USINT_TO_UDINT(exLink.StatsLastCall.minute) * 60000) + (USINT_TO_UDINT(exLink.StatsLastCall.second) * 1000));

			// Set stats timer
			Internal.StatsRefresh.IN := TRUE;
			Internal.StatsRefresh.PT := exLink.Configuration.CalculationTimeBase/10;
			Internal.StatsRefresh();

			// Internal data backup timer
			Internal.BackupTimer.IN := TRUE;
			Internal.BackupTimer.PT := CORE_BACKUP_TIMER*60*100;
			Internal.BackupTimer();
			IF Internal.BackupTimer.Q THEN
				Internal.BackupTimer.IN := FALSE;
				Internal.BackupTimer();

				Internal.State := exASSETINT_STATE_SAVE_LINK;
				RETURN;
			END_IF

			// Transfer downtime information
			Internal.Downtime := Downtime;
			IF ADR(DowntimeReason) <> 0 THEN
				Internal.DowntimeReason := DowntimeReason;
			ELSE
				Internal.DowntimeReason := '';
			END_IF

			// -------------------------------------------------------------------------------------------
			// Handle shift state change
			IF TrackShiftChange(ADR(exLink), ADR(Internal), ADR(Info), Parameters, Logger) THEN
				RETURN;
			END_IF

			// -------------------------------------------------------------------------------------------
			// Calculate shift and job statistics
			IF Internal.ShiftName <> '' THEN

				// Calculate new stats
				IF Internal.StatsRefresh.Q THEN
					// Get time difference between calls
					Internal.DiffLastCallShift := DiffT(clock_ms(), Internal.TimeLastCallShift);
					Internal.TimeLastCallShift := clock_ms();

					// Handle diff timer overflow
					IF Internal.DiffLastCallShift = 16#FFFFFFFF THEN
						CreateLoggerEntry(exASSETINT_LOG_INFO, ADR('diff timer overflow'), Logger);
					ELSE

						// Do not count when downtime is active
						IF Internal.Downtime = exASSETINT_NO_DOWNTIME THEN
							// Transfer job counter data
							IF Internal.JobPieceCounterOld <= PieceCounter THEN
								exLink.JobStatistics.TotalPieces := exLink.JobStatistics.TotalPieces + (PieceCounter - Internal.JobPieceCounterOld);
							ELSE
								CreateLoggerEntry(exASSETINT_LOG_ERROR, ADR('job piece count overflow'), Logger);
								exLink.JobStatistics.TotalPieces := exLink.JobStatistics.TotalPieces + (16#FFFFFFFF - Internal.JobPieceCounterOld + PieceCounter);
							END_IF

							IF Internal.JobRejectCounterOld <= RejectCounter THEN
								exLink.JobStatistics.RejectPieces := exLink.JobStatistics.RejectPieces + (RejectCounter - Internal.JobRejectCounterOld);
							ELSE
								CreateLoggerEntry(exASSETINT_LOG_ERROR, ADR('job reject count overflow'), Logger);
								exLink.JobStatistics.RejectPieces := exLink.JobStatistics.RejectPieces + (16#FFFFFFFF - Internal.JobRejectCounterOld + RejectCounter);
							END_IF
						END_IF
						Internal.JobPieceCounterOld := PieceCounter;
						Internal.JobRejectCounterOld := RejectCounter;
						CalcStatsJob(exLink, Internal.DiffLastCallShift, Internal.Downtime, Parameters, ADR(Info.JobStatistics));

						// Do not count when downtime is active
						IF Internal.Downtime = exASSETINT_NO_DOWNTIME THEN
							// Transfer shift counter data
							IF Internal.ShiftPieceCounterOld <= PieceCounter THEN
								exLink.ShiftStatistics.TotalPieces := exLink.ShiftStatistics.TotalPieces + (PieceCounter - Internal.ShiftPieceCounterOld);
							ELSE
								CreateLoggerEntry(exASSETINT_LOG_ERROR, ADR('shift piece count overflow'), Logger);
								exLink.ShiftStatistics.TotalPieces := exLink.ShiftStatistics.TotalPieces + (16#FFFFFFFF - Internal.ShiftPieceCounterOld + PieceCounter);
							END_IF

							IF Internal.ShiftRejectCounterOld <= RejectCounter THEN
								exLink.ShiftStatistics.RejectPieces := exLink.ShiftStatistics.RejectPieces + (RejectCounter - Internal.ShiftRejectCounterOld);
							ELSE
								CreateLoggerEntry(exASSETINT_LOG_ERROR, ADR('shift reject count overflow'), Logger);
								exLink.ShiftStatistics.RejectPieces := exLink.ShiftStatistics.RejectPieces + (16#FFFFFFFF - Internal.ShiftRejectCounterOld + RejectCounter);
							END_IF
						END_IF
						Internal.ShiftPieceCounterOld := PieceCounter;
						Internal.ShiftRejectCounterOld := RejectCounter;
						CalcStatsShift(exLink, Internal.DiffLastCallShift, Internal.Downtime, Parameters, ADR(Info.ShiftStatistics));

						// Transfer shift data to main function block
						CurrentProductionRate := exLink.ShiftStatistics.CurrentProductionRate;
						NominalProductionTimeRate := exLink.ShiftStatistics.NominalProductionTimeRate;
						BadPieceRate := exLink.ShiftStatistics.BadPieceRate;
						ScheduledDowntimeRate := exLink.ShiftStatistics.ScheduledDowntimeRate;
						UnscheduledDowntimeRate := exLink.ShiftStatistics.UnscheduledDowntimeRate;

					END_IF
				END_IF

				// When no shift is active
			ELSE
				// Dont count when no shift is active, reset last call
				Internal.ShiftPieceCounterOld := PieceCounter;
				Internal.ShiftRejectCounterOld := RejectCounter;
				Internal.JobPieceCounterOld := PieceCounter;
				Internal.JobRejectCounterOld := RejectCounter;

				Internal.TimeLastCallShift := clock_ms();
			END_IF

			// -------------------------------------------------------------------------------------------
			// Handle production state change
			IF TrackProductionState(ADR(exLink), ADR(Internal), Parameters, Logger) THEN
				RETURN;
			END_IF

			// -------------------------------------------------------------------------------------------
			// Handle update command
			IF EDGEPOS(Update) THEN
				CreateLoggerEntry(exASSETINT_LOG_INFO, ADR('update command triggered'), Logger);

				// -------------------------------------------------------------------------------------------
				// Check shift configuration for errors
				IF NOT exAssetIntCheckShiftData(Configuration, Logger, ADR(Internal.State), ADR(StatusID), ADR(Info.Diag.StatusID)) THEN
					RETURN;
				END_IF

				// Transfer configuration
				brsmemcpy(ADR(exLink.Configuration), ADR(Configuration), SIZEOF(Configuration));

				// Job has changed
				IF Parameters.Job <> exLink.JobStatistics.JobName THEN
					Internal.TmpStr1 := 'new job started ';
					brsstrcat(ADR(Internal.TmpStr1), ADR(Parameters.Job));
					CreateLoggerEntry(exASSETINT_LOG_INFO, ADR(Internal.TmpStr1), Logger);

					CommandBusy := TRUE;
					CommandDone := FALSE;
					UpdateDone := FALSE;

					// Transfer stats to record, make sure structures are allignent
					brsmemset(ADR(Internal.RecordData), 0, SIZEOF(Internal.RecordData));

					// Collect data for record
					Internal.RecordData.EventType := RecordTypeJob;
					Internal.RecordData.TimeStart := exLink.JobStatistics.StartTime;
					Internal.RecordData.TimeEnd := Internal.CurrentTime.DT1;
					// Take job user is known otherwise use current user from parameter
					IF exLink.JobStatistics.CurrentUser <> '' THEN
						Internal.RecordData.CurrentUser := exLink.JobStatistics.CurrentUser;
					ELSE
						Internal.RecordData.CurrentUser := Parameters.CurrentUser;
					END_IF
					Internal.RecordData.AdditionalData := Parameters.AdditionalData;
					Internal.RecordData.ShiftName := exLink.ShiftStatistics.ShiftName;
					Internal.RecordData.JobName := exLink.JobStatistics.JobName;
					Internal.RecordData.TotalPieces := exLink.JobStatistics.TotalPieces;
					Internal.RecordData.GoodPieces := exLink.JobStatistics.GoodPieces;
					Internal.RecordData.RejectPieces := exLink.JobStatistics.RejectPieces;
					Internal.RecordData.BadPieceRate := exLink.JobStatistics.BadPieceRate;
					Internal.RecordData.TotalTime := exLink.JobStatistics.TotalTime;
					Internal.RecordData.ScheduledDowntime := exLink.JobStatistics.ScheduledDowntime;
					Internal.RecordData.UnscheduledDowntime := exLink.JobStatistics.UnscheduledDowntime;
					Internal.RecordData.Uptime := exLink.JobStatistics.Uptime;
					Internal.RecordData.GoodProductionTime := exLink.JobStatistics.GoodProductionTime;
					Internal.RecordData.NominalProductionTime := exLink.JobStatistics.NominalProductionTime;
					Internal.RecordData.NominalProductionTimeRate := exLink.JobStatistics.NominalProductionTimeRate;
					Internal.RecordData.UnscheduledDowntimeRate := exLink.JobStatistics.UnscheduledDowntimeRate;
					Internal.RecordData.CurrentProductionRate := exLink.JobStatistics.CurrentProductionRate;

					// Reset stats and remember new start time
					brsmemset(ADR(Info.JobStatistics), 0, SIZEOF(Info.JobStatistics));
					brsmemset(ADR(exLink.JobStatistics), 0, SIZEOF(exLink.JobStatistics));

					exLink.JobTotalTime := 0;
					exLink.JobDowntimeScheduled := 0;
					exLink.JobDowntimeUnscheduled := 0;

					// Transfer data to job stats
					exLink.JobStatistics.StartTime := Internal.CurrentTime.DT1;
					exLink.JobStatistics.JobName := Parameters.Job;

					Internal.State := exASSETINT_STATE_STORE_EVENT;
				ELSE
					CommandBusy := FALSE;
					CommandDone := TRUE;
					UpdateDone := TRUE;
				END_IF

				// Transfer username and additional data
				exLink.JobStatistics.CurrentUser := Parameters.CurrentUser;
				exLink.JobStatistics.AdditionalData := Parameters.AdditionalData;

				exLink.ShiftStatistics.CurrentUser := Parameters.CurrentUser;
				exLink.ShiftStatistics.AdditionalData := Parameters.AdditionalData;

			END_IF

			IF NOT Update THEN
				UpdateDone := FALSE;
			END_IF

			// -------------------------------------------------------------------------------------------
			// Handle reset command
			IF EDGEPOS(Reset) THEN
				CreateLoggerEntry(exASSETINT_LOG_INFO, ADR('reset command triggered'), Logger);

				CommandBusy := TRUE;
				CommandDone := FALSE;

				// Reset stats
				brsmemset(ADR(Info.JobStatistics), 0, SIZEOF(Info.JobStatistics));
				brsmemset(ADR(exLink.JobStatistics), 0, SIZEOF(exLink.JobStatistics));

				exLink.JobTotalTime := 0;
				exLink.JobDowntimeScheduled := 0;
				exLink.JobDowntimeUnscheduled := 0;

				// Transfer data to job stats
				exLink.JobStatistics.StartTime := Internal.CurrentTime.DT1;
				exLink.JobStatistics.JobName := Parameters.Job;
				exLink.JobStatistics.CurrentUser := Parameters.CurrentUser;
				exLink.JobStatistics.AdditionalData := Parameters.AdditionalData;

				// Reset stats
				brsmemset(ADR(Info.ShiftStatistics), 0, SIZEOF(Info.ShiftStatistics));
				brsmemset(ADR(exLink.ShiftStatistics), 0, SIZEOF(exLink.ShiftStatistics));

				exLink.ShiftTotalTime := 0;
				exLink.ShiftDowntimeScheduled := 0;
				exLink.ShiftDowntimeUnscheduled := 0;

				// Transfer data to shift stats
				exLink.ShiftId := Internal.ShiftId;
				exLink.ShiftStatistics.StartTime := Internal.CurrentTime.DT1;
				exLink.ShiftStatistics.ShiftName := Internal.ShiftName;
				exLink.ShiftStatistics.CurrentUser := Parameters.CurrentUser;
				exLink.ShiftStatistics.AdditionalData := Parameters.AdditionalData;

				CommandBusy := FALSE;
				CommandDone := TRUE;
			END_IF

			// -------------------------------------------------------------------------------------------
			// Handle export command
			IF EDGEPOS(Export) THEN

				CommandBusy := TRUE;
				CommandDone := FALSE;
				ExportDone := FALSE;

				Internal.State := exASSETINT_STATE_EXPORT_EVENTS;
			END_IF

			IF NOT Export THEN
				ExportDone := FALSE;
			END_IF

			// -------------------------------------------------------------------------------------------
			// Reset refresh timer
			IF Internal.StatsRefresh.Q THEN
				// Set stats timer
				Internal.StatsRefresh.IN := FALSE;
				Internal.StatsRefresh();
			END_IF

			IF Update = FALSE AND Export = FALSE AND Reset = FALSE THEN
				CommandDone := FALSE;
			END_IF

			// -------------------------------------------------------------------------------------------
			// Store new event
			// -------------------------------------------------------------------------------------------
		exASSETINT_STATE_STORE_EVENT:
			// Find new record name
			IF exLink.RecordCount < CORE_EVENT_NUM_MAX THEN
				// Make sure record index is not already used
				FOR Internal.x := 0 TO exLink.RecordCount DO
					IF NOT Internal.RecordIndexUsed[Internal.x] THEN
						Internal.RecordIndex := Internal.x;
						EXIT;
					END_IF
				END_FOR;
			ELSE
				// Use last entry record name
				brsmemset(ADR(Internal.TmpStr1), 0, SIZEOF(Internal.TmpStr1));
				brsmemcpy(ADR(Internal.TmpStr1), exLink.MemoryDb + (exLink.RecordCount - 1)*SIZEOF(Internal.RecordData) +  1, SIZEOF(Internal.RecordData.FileName));
				brsstrcpy(ADR(Internal.TmpStr1), ADR(Internal.TmpStr1) + FindInstr(ADR(Internal.TmpStr1), ADR('#')) + 1);
				Internal.RecordIndex := DINT_TO_UINT(brsatoi(ADR(Internal.TmpStr1)));
				// Make sure parsed index stays within RecordIndexUsed
				IF Internal.RecordIndex > CORE_EVENT_NUM_MAX THEN
					Internal.RecordIndex := CORE_EVENT_NUM_MAX;
				END_IF
			END_IF

			Internal.WriteEventData.Enable := TRUE;
			Internal.WriteEventData.Device := StorageName;
			Internal.WriteEventData.Logger := Logger;
			Internal.WriteEventData.RecordData := ADR(Internal.RecordData);
			Internal.WriteEventData.RecordIndex := Internal.RecordIndex;
			Internal.WriteEventData();

			// -------------------------------------------------------------------------------------------
			// Event successful created
			IF Internal.WriteEventData.Status = ERR_OK THEN
				CreateLoggerEntry(exASSETINT_LOG_INFO, ADR('create new event ok'), Logger);

				// Copy new record into memeory
				IF exLink.RecordCount < CORE_EVENT_NUM_MAX THEN
					exLink.RecordCount := exLink.RecordCount + 1;
				END_IF
				brsmemmove(exLink.MemoryDb + SIZEOF(Internal.RecordData), exLink.MemoryDb, SIZEOF(Internal.RecordData)*(exLink.RecordCount - 1));
				brsmemcpy(exLink.MemoryDb, ADR(Internal.RecordData), SIZEOF(Internal.RecordData));
				Internal.RecordIndexUsed[Internal.RecordIndex] := TRUE;

				// Refrehs UI data, finish up
				exLink.RefreshJobUI := TRUE;
				exLink.RefreshShiftUI := TRUE;
				exLink.RefreshTimelineUI := TRUE;

				// Set update done flag
				IF Update AND CommandBusy THEN
					UpdateDone := TRUE;
				END_IF
				CommandBusy := FALSE;
				CommandDone := TRUE;

				StatusID := ERR_OK;
				Internal.State := exASSETINT_STATE_IDLE;

				// Error
			ELSIF Internal.WriteEventData.Status <> ERR_FUB_BUSY THEN
				// Set status, remember state, go to error state
				StatusID := CreateErrorState(Internal.WriteEventData.Status, ADR('ERR: create new event'), Logger, exCOM_SEV_ERROR, ADR(Internal.State), ADR(Info.Diag.StatusID));
			END_IF

			// -------------------------------------------------------------------------------------------
			// Export all events
			// -------------------------------------------------------------------------------------------
		exASSETINT_STATE_EXPORT_EVENTS:
			Internal.ExportEventData.Enable := TRUE;
			Internal.ExportEventData.Device := DeviceName;
			Internal.ExportEventData.Logger := Logger;
			Internal.ExportEventData.RecordCount := exLink.RecordCount;
			Internal.ExportEventData.Memory := exLink.MemoryDb;
			Internal.ExportEventData.Configuration := exLink.Configuration.Export;
			Internal.ExportEventData();

			// -------------------------------------------------------------------------------------------
			// Event successful created
			IF Internal.ExportEventData.Status = ERR_OK THEN
				CreateLoggerEntry(exASSETINT_LOG_INFO, ADR('export events ok'), Logger);

				ExportDone := TRUE;
				CommandBusy := FALSE;
				CommandDone := TRUE;

				StatusID := ERR_OK;
				Internal.State := exASSETINT_STATE_IDLE;

				// Error
			ELSIF Internal.ExportEventData.Status <> ERR_FUB_BUSY THEN
				// Set status, remember state, go to error state
				StatusID := CreateErrorState(Internal.ExportEventData.Status, ADR('ERR: export events'), Logger, exCOM_SEV_ERROR, ADR(Internal.State), ADR(Info.Diag.StatusID));
			END_IF

			// -------------------------------------------------------------------------------------------
			// Load link data
		exASSETINT_STATE_LOAD_LINK:
			Internal.ReadLinkData.Enable := TRUE;
			Internal.ReadLinkData.Device := ADR(StorageName);
			Internal.ReadLinkData.Logger := Logger;
			Internal.ReadLinkData.Link	 := ADR(exLink);
			Internal.ReadLinkData();

			// Link data successful restored
			IF Internal.ReadLinkData.Status = ERR_OK THEN
				CreateLoggerEntry(exASSETINT_LOG_INFO, ADR('load link data restored'), Logger);

				StatusID := ERR_OK;
				Internal.State := exASSETINT_STATE_INIT_2;

				// Link data does not exist
			ELSIF Internal.ReadLinkData.Status = fiERR_FILE_NOT_FOUND  THEN
				CreateLoggerEntry(exASSETINT_LOG_INFO, ADR('no backup file found'), Logger);

				StatusID := ERR_OK;
				Internal.State := exASSETINT_STATE_INIT_2;

				// Backup was corrupt (wrong size or version), it has already been deleted by ReadLinkData - start fresh
			ELSIF Internal.ReadLinkData.Status = ERR_ASSET_LINK_SIZE OR Internal.ReadLinkData.Status = ERR_ASSET_LINK_VERSION THEN
				CreateLoggerEntry(exASSETINT_LOG_INFO, ADR('corrupt backup file removed, starting fresh'), Logger);

				StatusID := ERR_OK;
				Internal.State := exASSETINT_STATE_INIT_2;

				// Error
			ELSIF Internal.ReadLinkData.Status <> ERR_FUB_BUSY THEN
				// Set status, remember state, go to error state
				StatusID := CreateErrorState(Internal.ReadLinkData.Status, ADR('ERR: load link data'), Logger, exCOM_SEV_ERROR,  ADR(Internal.State), ADR(Info.Diag.StatusID));
			END_IF

			// -------------------------------------------------------------------------------------------
			// Save link data
		exASSETINT_STATE_SAVE_LINK:
			Internal.WriteLinkData.Enable := TRUE;
			Internal.WriteLinkData.Device := ADR(StorageName);
			Internal.WriteLinkData.Logger := Logger;
			Internal.WriteLinkData.Link := ADR(exLink);
			Internal.WriteLinkData();

			// Event successful created
			IF Internal.WriteLinkData.Status = ERR_OK THEN
				CreateLoggerEntry(exASSETINT_LOG_INFO, ADR('save link data ok'), Logger);

				StatusID := ERR_OK;
				Internal.State := exASSETINT_STATE_IDLE;

				// Error
			ELSIF Internal.WriteLinkData.Status <> ERR_FUB_BUSY THEN
				// Set status, remember state, go to error state
				StatusID := CreateErrorState(Internal.WriteLinkData.Status, ADR('ERR: save link data'), Logger, exCOM_SEV_ERROR,  ADR(Internal.State), ADR(Info.Diag.StatusID));
			END_IF

			// -------------------------------------------------------------------------------------------
			// Error state
			// -------------------------------------------------------------------------------------------
		exASSETINT_STATE_ERROR:
			Error := TRUE;

			// Reset error state
			IF EDGEPOS(ErrorReset) THEN
				Internal.StateError := exASSETINT_STATE_NONE;
				Internal.State := exASSETINT_STATE_INIT_1;
			END_IF
	END_CASE;

END_FUNCTION_BLOCK
```
